FUNCTION_BLOCK HigherLevelFB EXTENDS SignalHandling
VAR_INPUT
END_VAR
VAR_OUTPUT
END_VAR
VAR
	fbTest : TESTFB;
	stException : ST_Exception;
	bSystemException : BOOL;
	bWrongValueException : BOOL;
END_VAR

SUPER^();
fbTest(eOrigin := eTEST_UNIT);

IF fbTest.Catch(eWRONG_VALUE_EXCEPTION, fbTest.getExceptionOrigin) 
THEN
	;
// React to error here
// Catch must reset the exception in fbTest
	bWrongValueException := TRUE;	
END_IF

//Forward all other exceptions to the next higher level
IF fbTest.ExceptionAvailable()
THEN

	//ForwardToNextLevel must set all exceptions in fbTest on forwarded
	ForwardToNextLevel(fbTest);
	
END_IF

IF bSystemException
THEN
	Throw(BuildException(eSYSTEM_EXCEPTION));
END_IF

END_FUNCTION_BLOCK

(* stored: Version 1.1.0.1, ProductVersion 3.1.4024.0
   POU HigherLevelFB: Id {b72c46aa-1dd1-419c-8ff8-f3de5d8c59b9}, SpecialFunc None *)
